TYPE ST_OEE_Out :
STRUCT
	Quality												: REAL;
	Performance											: REAL;
	Availability										: REAL;
	OEE													: REAL;
	Active												: BOOL;
	EnableOut											: BOOL;	
END_STRUCT
END_TYPE

(* stored: Version 1.1.0.1, ProductVersion 3.1.4024.2
   DUT ST_OEE_Out: Id {4b49f4af-8f3a-4edd-a391-fb0c4594b0c8} *)
